Fanuc KAREL source: kc00022.KL

-- PROVISIONAL review KL for V770-1; original PC SHA256 61d7bac5e21ff59ecf5043fa8aae08edce5133bc8620254bc3122bcdbf05f819
-- Incomplete behavior may be omitted. Consult companion uncertainty JSON. Do not deploy.
PROGRAM KC00022
%NOLOCKGROUP
BEGIN
  -- UNRESOLVED_PC offsets 5-22; opcodes 3F,75
  -- UNRESOLVED_PC offsets 27-45; opcodes 27,22,2A,22,31
  -- UNRESOLVED_PC offsets 50-54; opcodes 7F
END KC00022
